Omron Sysmac Studio project modbus_tcpip_hmi_server_nx1p2_client (Sysmac Studio 1.45.1.64010, StandardProject)

# Controller new_Controller_0: NX1P2-9024DT version 1.40
Units and slaves: Node86 : NX-ECC201 (E001); Unit 1 : NX-OD5121 (N1); Unit 2 : NX-OD4256 (N2); Unit 3 : NX-ID5342 (N3); Unit 4 : NX-ID5442 (N4); Node1 : GX-ID1611+OD16 (E002)
Task PrimaryTask (priority 4, period or condition 2000): Program0
Library OEN_Communication_V1_0_22 1.0.22 (contents left out)

VAR_GLOBAL
    start_hmi : BOOL;  (* published *)
    stop_hmi : BOOL;  (* published *)
    dong_co : BOOL;  (* published *)
    GX_OUT_0 : BOOL;  (* GX_WWXT_OD16; at ECAT://node#1/Write output 1st word/Out Bit00 *)
    GX_OUT_1 : BOOL;  (* GX_WWXT_OD16; at ECAT://node#1/Write output 1st word/Out Bit01 *)
    GX_OUT_2 : BOOL;  (* GX_WWXT_OD16; at ECAT://node#1/Write output 1st word/Out Bit02 *)
    GX_OUT_3 : BOOL;  (* GX_WWXT_OD16; at ECAT://node#1/Write output 1st word/Out Bit03 *)
    GX_OUT_4 : BOOL;  (* GX_WWXT_OD16; at ECAT://node#1/Write output 1st word/Out Bit04 *)
    GX_OUT_5 : BOOL;  (* GX_WWXT_OD16; at ECAT://node#1/Write output 1st word/Out Bit05 *)
    GX_OUT_6 : BOOL;  (* GX_WWXT_OD16; at ECAT://node#1/Write output 1st word/Out Bit06 *)
    GX_OUT_7 : BOOL;  (* GX_WWXT_OD16; at ECAT://node#1/Write output 1st word/Out Bit07 *)
    GX_OUT_8 : BOOL;  (* GX_WWXT_OD16; at ECAT://node#1/Write output 1st word/Out Bit08 *)
    GX_OUT_9 : BOOL;  (* GX_WWXT_OD16; at ECAT://node#1/Write output 1st word/Out Bit09 *)
    GX_OUT_10 : BOOL;  (* GX_WWXT_OD16; at ECAT://node#1/Write output 1st word/Out Bit10 *)
    GX_OUT_11 : BOOL;  (* GX_WWXT_OD16; at ECAT://node#1/Write output 1st word/Out Bit11 *)
    GX_OUT_12 : BOOL;  (* GX_WWXT_OD16; at ECAT://node#1/Write output 1st word/Out Bit12 *)
    GX_OUT_13 : BOOL;  (* GX_WWXT_OD16; at ECAT://node#1/Write output 1st word/Out Bit13 *)
    GX_OUT_14 : BOOL;  (* GX_WWXT_OD16; at ECAT://node#1/Write output 1st word/Out Bit14 *)
    GX_OUT_15 : BOOL;  (* GX_WWXT_OD16; at ECAT://node#1/Write output 1st word/Out Bit15 *)
    OD5121_OUT_0 : BOOL;  (* NX_ECC201_MD_OD5121_NPN; at ECAT://node#[86,1]/Output Bit 16 bits/Output Bit 00 *)
    OD5121_OUT_1 : BOOL;  (* NX_ECC201_MD_OD5121_NPN; at ECAT://node#[86,1]/Output Bit 16 bits/Output Bit 01 *)
    OD5121_OUT_2 : BOOL;  (* NX_ECC201_MD_OD5121_NPN; at ECAT://node#[86,1]/Output Bit 16 bits/Output Bit 02 *)
    OD5121_OUT_3 : BOOL;  (* NX_ECC201_MD_OD5121_NPN; at ECAT://node#[86,1]/Output Bit 16 bits/Output Bit 03 *)
    OD5121_OUT_4 : BOOL;  (* NX_ECC201_MD_OD5121_NPN; at ECAT://node#[86,1]/Output Bit 16 bits/Output Bit 04 *)
    OD5121_OUT_5 : BOOL;  (* NX_ECC201_MD_OD5121_NPN; at ECAT://node#[86,1]/Output Bit 16 bits/Output Bit 05 *)
    OD5121_OUT_6 : BOOL;  (* NX_ECC201_MD_OD5121_NPN; at ECAT://node#[86,1]/Output Bit 16 bits/Output Bit 06 *)
    OD5121_OUT_7 : BOOL;  (* NX_ECC201_MD_OD5121_NPN; at ECAT://node#[86,1]/Output Bit 16 bits/Output Bit 07 *)
    OD5121_OUT_8 : BOOL;  (* NX_ECC201_MD_OD5121_NPN; at ECAT://node#[86,1]/Output Bit 16 bits/Output Bit 08 *)
    OD5121_OUT_9 : BOOL;  (* NX_ECC201_MD_OD5121_NPN; at ECAT://node#[86,1]/Output Bit 16 bits/Output Bit 09 *)
    OD5121_OUT_10 : BOOL;  (* NX_ECC201_MD_OD5121_NPN; at ECAT://node#[86,1]/Output Bit 16 bits/Output Bit 10 *)
    OD5121_OUT_11 : BOOL;  (* NX_ECC201_MD_OD5121_NPN; at ECAT://node#[86,1]/Output Bit 16 bits/Output Bit 11 *)
    OD5121_OUT_12 : BOOL;  (* NX_ECC201_MD_OD5121_NPN; at ECAT://node#[86,1]/Output Bit 16 bits/Output Bit 12 *)
    OD5121_OUT_13 : BOOL;  (* NX_ECC201_MD_OD5121_NPN; at ECAT://node#[86,1]/Output Bit 16 bits/Output Bit 13 *)
    OD5121_OUT_14 : BOOL;  (* NX_ECC201_MD_OD5121_NPN; at ECAT://node#[86,1]/Output Bit 16 bits/Output Bit 14 *)
    OD5121_OUT_15 : BOOL;  (* NX_ECC201_MD_OD5121_NPN; at ECAT://node#[86,1]/Output Bit 16 bits/Output Bit 15 *)
    NX1P2_OUT_0 : BOOL;  (* NX1P2_9024DT_OUT; at BuiltInIO://cpu/#0/Output_Bit_00 *)
    NX1P2_OUT_1 : BOOL;  (* NX1P2_9024DT_OUT; at BuiltInIO://cpu/#0/Output_Bit_01 *)
    NX1P2_OUT_2 : BOOL;  (* NX1P2_9024DT_OUT; at BuiltInIO://cpu/#0/Output_Bit_02 *)
    NX1P2_OUT_3 : BOOL;  (* NX1P2_9024DT_OUT; at BuiltInIO://cpu/#0/Output_Bit_03 *)
    NX1P2_OUT_4 : BOOL;  (* NX1P2_9024DT_OUT; at BuiltInIO://cpu/#0/Output_Bit_04 *)
    NX1P2_OUT_5 : BOOL;  (* NX1P2_9024DT_OUT; at BuiltInIO://cpu/#0/Output_Bit_05 *)
    NX1P2_OUT_6 : BOOL;  (* NX1P2_9024DT_OUT; at BuiltInIO://cpu/#0/Output_Bit_06 *)
    NX1P2_OUT_7 : BOOL;  (* NX1P2_9024DT_OUT; at BuiltInIO://cpu/#0/Output_Bit_07 *)
    NX1P2_OUT_8 : BOOL;  (* NX1P2_9024DT_OUT; at BuiltInIO://cpu/#0/Output_Bit_08 *)
    NX1P2_OUT_9 : BOOL;  (* NX1P2_9024DT_OUT; at BuiltInIO://cpu/#0/Output_Bit_09 *)
    OD5121_REGISTER : WORD;  (* NX_ECC201_MD_OD5121_NPN; at ECAT://node#[86,1]/Output Bit 16 bits *)
    REGISTER_GX_OUT : WORD;  (* GX_WWXT_OD16; at ECAT://node#1/Write output 1st word *)
END_VAR

PROGRAM Program0
VAR
    DISCONNECT_TCP_CLIENT : BOOL;
    TCP_CLIENT_CONNECT : BOOL;
    T_CONNECT_TCP : TON;
    T_CONNECT_TCP_CLIENT : TON;
    MODBUS_CLIENT : OEN\Modbus\ModbusTCP_Client;
    REQUEST_CLIENT : ARRAY[0..3] OF OEN\Modbus\sModbusReq := [(Enable := True, NodeAdr := 0, FunctionCode := Fn03_ReadHoldingRegisters, Read := (StartAddressRemote := 0, StartAddressLocal := 0, Count := 4), Write := (StartAddressRemote := 0, StartAddressLocal := 0, Count := 0)), (Enable := True, NodeAdr := 0, FunctionCode := Fn16_WriteMultipleRegisters, Read := (StartAddressRemote := 0, StartAddressLocal := 0, Count := 0), Write := (StartAddressRemote := 4, StartAddressLocal := 4, Count := 6)), (Enable := True, NodeAdr := 0, FunctionCode := Fn03_ReadHoldingRegisters, Read := (StartAddressRemote := 10, StartAddressLocal := 10, Count := 7), Write := (StartAddressRemote := 0, StartAddressLocal := 0, Count := 0)), (Enable := True, NodeAdr := 0, FunctionCode := Fn16_WriteMultipleRegisters, Read := (StartAddressRemote := 0, StartAddressLocal := 0, Count := 0), Write := (StartAddressRemote := 17, StartAddressLocal := 17, Count := 6))];
    DATA_COIL_CLIENT : ARRAY[0..16] OF BOOL;
    DISCRETELINPUT_CLIENT : ARRAY[0..16] OF BOOL;
    INPUT_REGISTER_CLIENT : ARRAY[0..16] OF WORD;
    HOLDINGREGISTERR_CLIENT : ARRAY[0..31] OF WORD;
    REQUEST_DONE : BOOL;
    REQUEST_CLYCLE_TIME : TIME;
    TCP_CONNECT : BOOL;
    DATA_WRITE_0 : WORD;
    DATA_WRITE_1 : WORD;
    DATA_WRITE_2 : WORD;
    DATA_WRITE_3 : WORD;
    DATA_WRITE_4 AT %W0 : WORD;
    DATA_WRITE_5 : WORD;
    INT_DATA_WRITE_5 : INT;
    INT_WRITE_4 : INT;
    DINT_DATA_WRITE_6 : DINT;
    INT_DATA_READ_4 : INT;
    INT_DATA_READ_0 : INT;
    INT_DATA_READ_1 : DINT;
    INT_DATA_READ_5 : INT;
    INT_DATA_READ_6 : INT;
    INT_DATA_LOW_READ_5 : INT;
    INT_DATA_HIGH_READ_5 : INT;
    INT_DATA_READ_7 : INT;
    DISCONNECT_MODBUS_TCP_CLIENT : BOOL;
    VAL_CONTROL_OD1611 : DWORD;
    VAL_TRGIAN_RES_01 : WORD;
    INT_DATA_CONTROL : DINT;
    INT_HIGH_RES_DWORD_0 : DINT;
    OUT : BOOL;
    DATA_READ_12 : WORD;
    DATA_READ_13 : WORD;
    REGISTER_12 : DINT;
    T_COUNT_1 : TON;
    DATA_READ_4 : WORD;
    COUNT_1 : INT;
END_VAR
VAR RETAIN
    SV_COUNT_1 : int;
END_VAR
VAR
    T_COUNT_2 : TON;
    H : INT;
END_VAR
VAR RETAIN
    DATA_RES_15 AT %D15 : WORD;
END_VAR
VAR
    T1 : TON;
    T2 : TON;
    km_1 : int;
    km_3 : int;
    km_4 : int;
    reading_array_1 : ARRAY[0..2] OF int;
    reading_array_2 : ARRAY[0..6] OF int;
    write_array_2 : ARRAY[0..5] OF int;
    write_array_3 : ARRAY[0..5] OF int;
    km_2 : int;
END_VAR
VAR_EXTERNAL
    start_hmi : BOOL;
    dong_co : BOOL;
    stop_hmi : BOOL;
    NX1P2_OUT_0 : BOOL;
    REGISTER_GX_OUT : WORD;
END_VAR

(* Section connect_modbus_client: ladder, written here as Structured Text *)

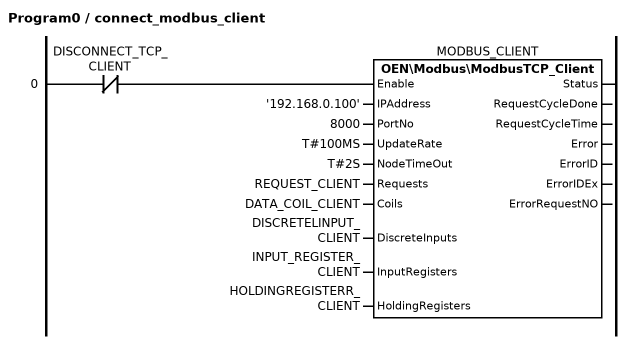
(* Rung 0 *)
MODBUS_CLIENT(Enable := NOT DISCONNECT_TCP_CLIENT, IPAddress := '192.168.0.100', PortNo := 8000, UpdateRate := T#100MS, NodeTimeOut := T#2S, Requests := REQUEST_CLIENT, Coils := DATA_COIL_CLIENT, DiscreteInputs := DISCRETELINPUT_CLIENT, InputRegisters := INPUT_REGISTER_CLIENT, HoldingRegisters := HOLDINGREGISTERR_CLIENT);

(* Section read_data_hmi: ladder, written here as Structured Text *)

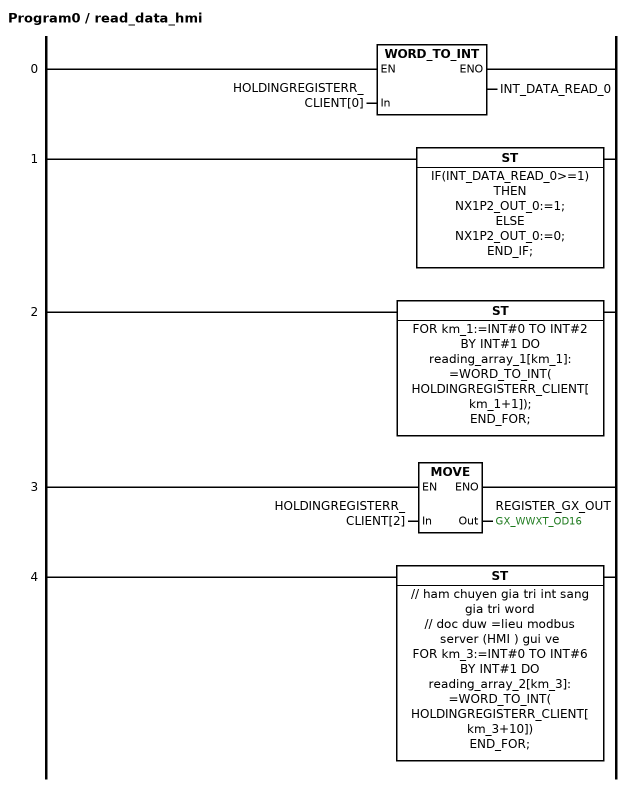
(* Rung 0 *)
INT_DATA_READ_0 := WORD_TO_INT(In := HOLDINGREGISTERR_CLIENT[0]);
(* Rung 1 *)
IF(INT_DATA_READ_0>=1) THEN
	NX1P2_OUT_0:=1;
ELSE
	NX1P2_OUT_0:=0;
END_IF;
(* Rung 2 *)
FOR km_1:=INT#0 TO INT#2 BY INT#1 DO
  reading_array_1[km_1]:=WORD_TO_INT(HOLDINGREGISTERR_CLIENT[km_1+1]);
END_FOR;
(* Rung 3 *)
REGISTER_GX_OUT := HOLDINGREGISTERR_CLIENT[2];
(* Rung 4 *)
 // ham chuyen gia tri int sang gia tri word
 // doc duw =lieu modbus server (HMI ) gui ve
FOR km_3:=INT#0 TO INT#6 BY INT#1 DO
  reading_array_2[km_3]:=WORD_TO_INT(HOLDINGREGISTERR_CLIENT[km_3+10]);
END_FOR;

(* Section write_data_hmi: ladder, written here as Structured Text *)

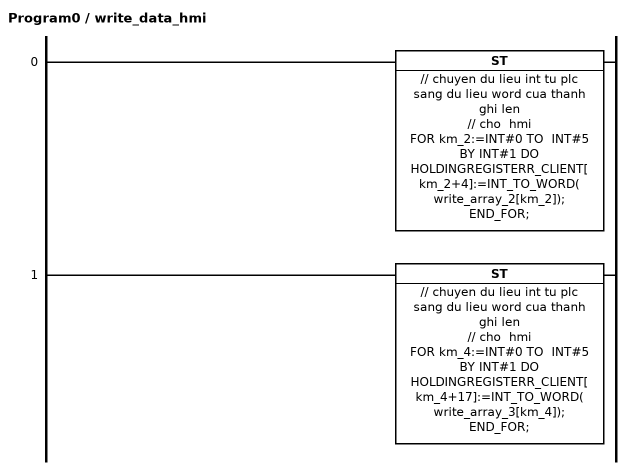
(* Rung 0 *)
// chuyen du lieu int tu plc sang du lieu word cua thanh ghi len
// cho  hmi
FOR km_2:=INT#0 TO  INT#5 BY INT#1 DO
	 HOLDINGREGISTERR_CLIENT[km_2+4]:=INT_TO_WORD(write_array_2[km_2]);
END_FOR;
(* Rung 1 *)
// chuyen du lieu int tu plc sang du lieu word cua thanh ghi len
// cho  hmi
FOR km_4:=INT#0 TO  INT#5 BY INT#1 DO
	 HOLDINGREGISTERR_CLIENT[km_4+17]:=INT_TO_WORD(write_array_3[km_4]);
END_FOR;
END_PROGRAM